Staubli VAL3: TxtReadRoom1.pgx

program TxtReadRoom1()
  local num l_ntest
  local num l_n
begin
  delay(0.01)
  l_ntest=$fileOpen(sTxtfile[n_sTxt],"r")
  for l_n=0 to 499
    $fileGet(l_ntest,sString[l_n],1)
    if sString[l_n]!=""
      call stringtopoint(sString[l_n],l_n)
    else
    endIf
  endFor
  delay(0.01)
  bTxt1=false
  if n_sTxt==nTxtTotal-1
    n_sTxt=0
  else
    n_sTxt=n_sTxt+1
  endIf

  $fileClose(l_ntest)
  call hmi_refreshmain()
end
